// TIA Portal project "Projekt_magazyn" (V13)
// Vorlageprojekt für das Buch mit Zielsystem S7-1200

(* hardware
DEVICE "S7-1200-Station_1"  S7-1200 Station
   slot 0: "Baugruppenträger_0"  Rack  V1.0
   slot 1: "PLC_1"  CPU 1211C DC/DC/DC  6ES7 211-1AE40-0XB0  V4.1
*)

// ===== PLC "PLC_1"  CPU 1211C DC/DC/DC =====

VAR_GLOBAL   // PLC tag table "Wejścia"
   "Start" AT %I10.0 : Bool;
   "Reset" AT %I10.1 : Bool;
   "Stop" AT %I10.2 : Bool;
   "Manual" AT %I10.3 : Bool;
   "Auto" AT %I10.4 : Bool;
   "Emergency stop" AT %I10.5 : Bool;
   "Stop Baza 1" AT %I10.6 : Bool;
   "Czujnik KUKA Baza" AT %I10.7 : Bool;
   "Czujnik Baza 1" AT %I11.0 : Bool;
   "Czujnik Stop Baza" AT %I11.1 : Bool;
   "Baza gotowa" AT %I11.2 : Bool;
   "Czujnik Zacisk Baza" AT %I11.3 : Bool;
   "Stop Pokrywa 1" AT %I11.4 : Bool;
   "Czujnik KUKA Pokrywa" AT %I11.5 : Bool;
   "Czujnik Pokrywa 1" AT %I11.6 : Bool;
   "Czujnik Stop POKRYWA" AT %I11.7 : Bool;
   "Pokrywa gotowa" AT %I12.0 : Bool;
   "Czujnik Zacisk POKRYWA" AT %I12.1 : Bool;
   "Pokrywa wykryta" AT %I12.2 : Bool;
   "Moving X" AT %I12.3 : Bool;
   "Moving Z" AT %I12.4 : Bool;
   "Pos. at limit (base)" AT %I12.5 : Bool;
   "Pos. at limit (lids)" AT %I12.6 : Bool;
   "FACTORY I/O (Running)" AT %I13.0 : Bool;
   "Czujnik Sortowania" AT %ID30 : DInt;
   "Czujnik Wyjscia" AT %I13.1 : Bool;
END_VAR

VAR_GLOBAL   // PLC tag table "Wyjścia"
   "Emiter BAZA" AT %Q0.0 : Bool;
   "Baza 1" AT %Q0.1 : Bool;
   "Kuka BAZA (Start)" AT %Q0.2 : Bool;
   "Kuka BAZA (Reset)" AT %Q0.3 : Bool;
   "Kuka BAZA (Produce Base)" AT %Q0.5 : Bool;
   "Kuka BAZA (Stop)" AT %Q0.4 : Bool;
   "Baza 2" AT %Q0.6 : Bool;
   "Stop BAZA" AT %Q0.7 : Bool;
   "Baza 3" AT %Q1.0 : Bool;
   "Baza 4" AT %Q1.1 : Bool;
   "Baza 5" AT %Q1.2 : Bool;
   "Emiter POKRYWA" AT %Q1.3 : Bool;
   "Pokrywa 1" AT %Q1.4 : Bool;
   "Kuka POKRYWA (Start)" AT %Q1.5 : Bool;
   "Kuka POKRYWA (Reset)" AT %Q1.6 : Bool;
   "Kuka POKRYWA (Stop)" AT %Q1.7 : Bool;
   "Kuka POKRYWA (Produce Lids)" AT %Q2.0 : Bool;
   "Pokrywa 2" AT %Q2.1 : Bool;
   "Stop POKRYWA" AT %Q2.2 : Bool;
   "Pokrywa 3" AT %Q2.3 : Bool;
   "Pokrywa 4" AT %Q2.4 : Bool;
   "Pokrywa 5" AT %Q2.5 : Bool;
   "Baza Assembler" AT %Q2.6 : Bool;
   "Pokrywa Assembler" AT %Q2.7 : Bool;
   "Zacisk POKRYWA" AT %Q3.1 : Bool;
   "Zlap" AT %Q3.2 : Bool;
   "Podnies BAZA" AT %Q3.3 : Bool;
   "Move Z" AT %Q3.5 : Bool;
   "Move X" AT %Q3.4 : Bool;
   "tasma 1" AT %Q3.6 : Bool;
   "tasma 2" AT %Q3.7 : Bool;
   "Ramie N" AT %Q4.0 : Bool;
   "Tasma Ramie N" AT %Q4.1 : Bool;
   "Ramie Z" AT %Q4.2 : Bool;
   "Tasma Ramie Z" AT %Q4.3 : Bool;
   "Ramie I" AT %Q4.4 : Bool;
   "Tasma Ramie I" AT %Q4.5 : Bool;
   "NIEBIESKIE" AT %Q4.6 : Bool;
   "ZIELONE" AT %Q4.7 : Bool;
   "INNE" AT %Q5.0 : Bool;
   "Start light" AT %Q5.1 : Bool;
   "Reset light" AT %Q5.2 : Bool;
   "Stop light" AT %Q5.3 : Bool;
   "Zacisk BAZA" AT %Q3.0 : Bool;
   "Licznik Zielone" AT %QD34 : DInt;
   "Licznik Niebieskie" AT %QD30 : DInt;
   "Licznik Inne" AT %QD38 : DInt;
END_VAR

VAR_GLOBAL   // PLC tag table "Markery"
   "M0" AT %M0.0 : Bool;
   "M1" AT %M0.1 : Bool;
   "M2" AT %M0.2 : Bool;
   "M3" AT %M0.3 : Bool;
   "M4" AT %M0.4 : Bool;
   "M5" AT %M0.5 : Bool;
   "M6" AT %M0.6 : Bool;
   "Czujnik Sortowania w zakresie" AT %M1.4 : Bool;
   "Always False" AT %M2.0 : Bool;
END_VAR

// folder: System blocks/Program resources

DATA_BLOCK "IEC_Counter_0_DB"   // DB2
{ S7_Optimized_Access := 'FALSE' }
AUTHOR : Simatic
FAMILY : IEC
NAME : CNTR
VERSION : 1.0
// stored: InstanceOfName ?
"?"
BEGIN
END_DATA_BLOCK

DATA_BLOCK "IEC_Counter_0_DB_1"   // DB3
{ S7_Optimized_Access := 'FALSE' }
AUTHOR : Simatic
FAMILY : IEC
NAME : CNTR
VERSION : 1.0
// stored: InstanceOfName ?
"?"
BEGIN
END_DATA_BLOCK

DATA_BLOCK "IEC_Counter_0_DB_2"   // DB4
{ S7_Optimized_Access := 'FALSE' }
AUTHOR : Simatic
FAMILY : IEC
NAME : CNTR
VERSION : 1.0
// stored: InstanceOfName ?
"?"
BEGIN
END_DATA_BLOCK

// folder: (top level)

FUNCTION "MHJ-PLC-Lab-Function-S71200" : Void   // FC9000, SCL
{ S7_Optimized_Access := 'FALSE' }
VERSION : 0.1
BEGIN

   #Value:=PEEK(area := 16#82,
        dbNumber := 0,
        byteOffset := 511);
   #Value := #Value + 1;

   POKE(area := 16#82,
        dbNumber := 0,
        byteOffset := 511,
        value := #Value);

   POKE(area:=16#81,
        dbNumber:=0,
        byteOffset:=1016,
        value:=#Value_01_DW);
   POKE(area := 16#81,
        dbNumber := 0,
        byteOffset := 1020,
        value := #Value_02_DW);

   POKE(area := 16#81,
        dbNumber := 0,
        byteOffset := 511,
        value := B#16#00);

   FOR #forVal := 0 TO 120 DO
       FOR #forVal_2:=0 TO 10 DO
           #rdTimeReturn:=RD_SYS_T(#outputTime);
           #rdTimeReturn := WR_SYS_T(#outputTime);
           #rdTimeReturn := RD_SYS_T(#outputTime);
           #rdTimeReturn := WR_SYS_T(#outputTime);
       END_FOR;
       #SyncVal:= PEEK(area := 16#81,
                      dbNumber := 0,
                      byteOffset := 511);
       IF #SyncVal = #CompVal THEN
          GOTO M_1;
       END_IF;
   END_FOR;
   RETURN;

   M_1:
   POKE(area := 16#81,
        dbNumber := 0,
        byteOffset := 511,
        value := B#16#0);
END_FUNCTION

ORGANIZATION_BLOCK "Sortownia"   // OB1, LAD, ProgramCycle
TITLE = "Main Program Sweep (Cycle)"
{ S7_Optimized_Access := 'FALSE' }
VERSION : 0.1
   VAR_TEMP   // added for the SCL form of the ladder/FBD networks
      _w1 : Bool;
   END_VAR
BEGIN

REGION Network 1
   // Czujnik Sortowania (zakres wykrywania pokrywek według dokumentacji Factory IO)
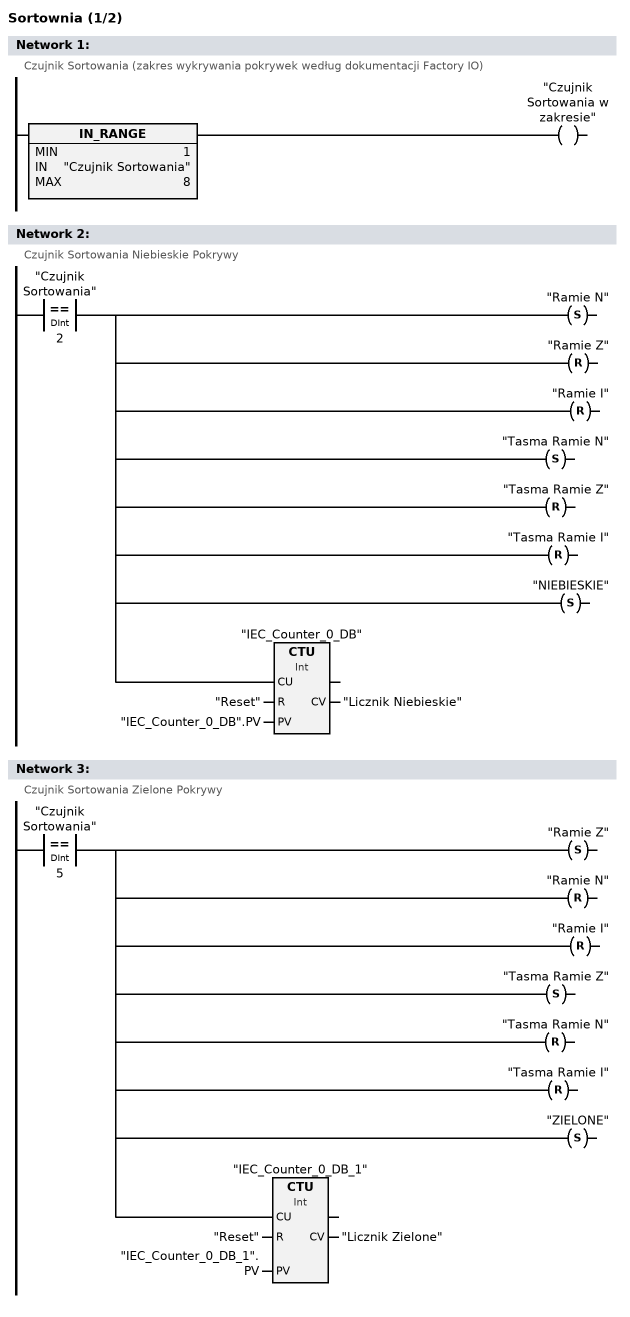
   RUNG wire#powerrail
      { S7_Templates := "SrcType := DInt" } InRange(min := 1, in := "Czujnik Sortowania", max := 8)
      Coil( "Czujnik Sortowania w zakresie" )
   END_RUNG
   // the same network as SCL:
   "Czujnik Sortowania w zakresie" := (1 <= "Czujnik Sortowania") AND ("Czujnik Sortowania" <= 8);
END_REGION

REGION Network 2
   // Czujnik Sortowania Niebieskie Pokrywy
   #_w1 := "Czujnik Sortowania" = 2;
   IF #_w1 THEN
       "Ramie N" := TRUE;
       "Ramie Z" := FALSE;
       "Ramie I" := FALSE;
       "Tasma Ramie N" := TRUE;
       "Tasma Ramie Z" := FALSE;
       "Tasma Ramie I" := FALSE;
       "NIEBIESKIE" := TRUE;
   END_IF;
   "IEC_Counter_0_DB".CTU(CU := #_w1, R := "Reset", PV := "IEC_Counter_0_DB".PV, CV => "Licznik Niebieskie");
END_REGION

REGION Network 3
   // Czujnik Sortowania Zielone Pokrywy
   #_w1 := "Czujnik Sortowania" = 5;
   IF #_w1 THEN
       "Ramie Z" := TRUE;
       "Ramie N" := FALSE;
       "Ramie I" := FALSE;
       "Tasma Ramie Z" := TRUE;
       "Tasma Ramie N" := FALSE;
       "Tasma Ramie I" := FALSE;
       "ZIELONE" := TRUE;
   END_IF;
   "IEC_Counter_0_DB_1".CTU(CU := #_w1, R := "Reset", PV := "IEC_Counter_0_DB_1".PV, CV => "Licznik Zielone");
END_REGION

REGION Network 4
   // Czujnik Sortowania Metalowe Pokrywy
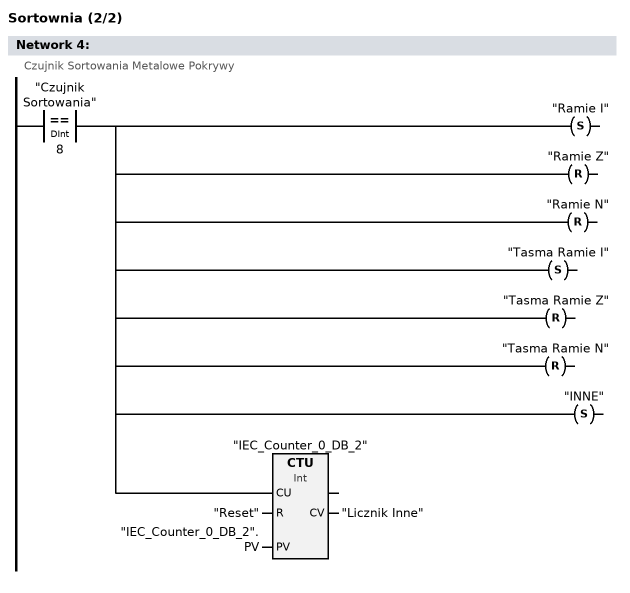
   #_w1 := "Czujnik Sortowania" = 8;
   IF #_w1 THEN
       "Ramie I" := TRUE;
       "Ramie Z" := FALSE;
       "Ramie N" := FALSE;
       "Tasma Ramie I" := TRUE;
       "Tasma Ramie Z" := FALSE;
       "Tasma Ramie N" := FALSE;
       "INNE" := TRUE;
   END_IF;
   "IEC_Counter_0_DB_2".CTU(CU := #_w1, R := "Reset", PV := "IEC_Counter_0_DB_2".PV, CV => "Licznik Inne");
END_REGION
END_ORGANIZATION_BLOCK

ORGANIZATION_BLOCK "Main 1"   // OB123, LAD, ProgramCycle
TITLE = "Main Program Sweep (Cycle)"
{ S7_Optimized_Access := 'FALSE' }
VERSION : 0.1
BEGIN

REGION Network 1
   // konfiguracja z Factory IO
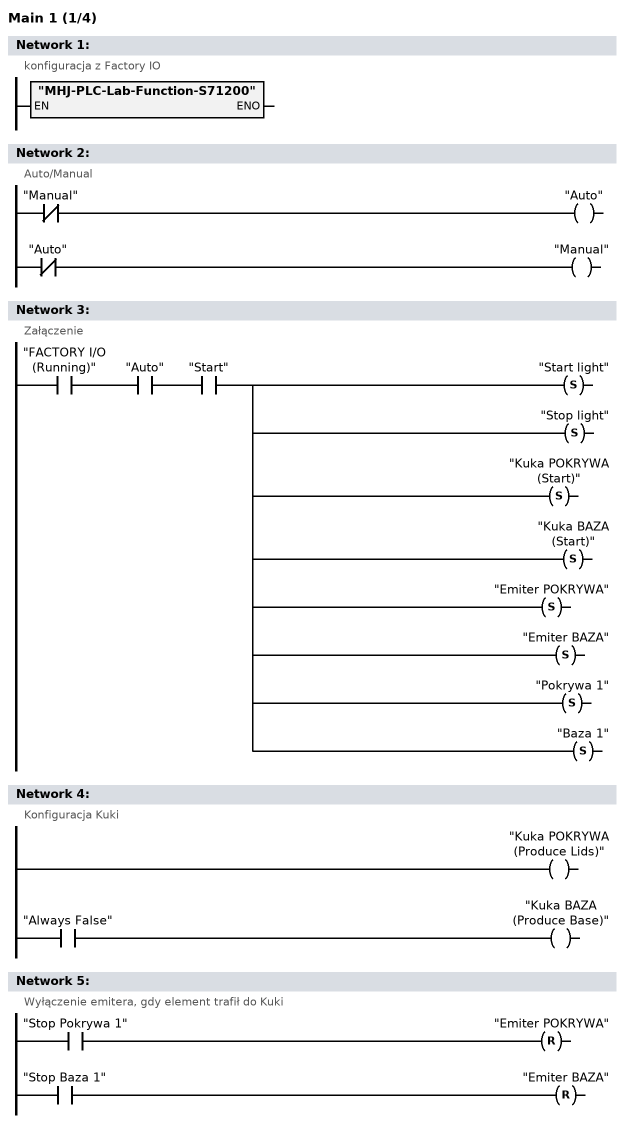
   RUNG wire#powerrail
      "MHJ-PLC-Lab-Function-S71200"()
   END_RUNG
   // the same network as SCL:
   "MHJ-PLC-Lab-Function-S71200"();
END_REGION

REGION Network 2
   // Auto/Manual
   RUNG wire#powerrail
      I_Contact( "Manual" )
      Coil( "Auto" )
   END_RUNG
   RUNG wire#powerrail
      I_Contact( "Auto" )
      Coil( "Manual" )
   END_RUNG
   // the same network as SCL:
   "Auto" := NOT "Manual";
   "Manual" := NOT "Auto";
END_REGION

REGION Network 3
   // Załączenie
   RUNG wire#powerrail
      Contact( "FACTORY I/O (Running)" )
      Contact( "Auto" )
      Contact( "Start" )
      wire#w1
      S_Coil( "Start light" )
   END_RUNG
   RUNG wire#w1
      S_Coil( "Stop light" )
   END_RUNG
   RUNG wire#w1
      S_Coil( "Kuka POKRYWA (Start)" )
   END_RUNG
   RUNG wire#w1
      S_Coil( "Kuka BAZA (Start)" )
   END_RUNG
   RUNG wire#w1
      S_Coil( "Emiter POKRYWA" )
   END_RUNG
   RUNG wire#w1
      S_Coil( "Emiter BAZA" )
   END_RUNG
   RUNG wire#w1
      S_Coil( "Pokrywa 1" )
   END_RUNG
   RUNG wire#w1
      S_Coil( "Baza 1" )
   END_RUNG
   // the same network as SCL:
   IF "FACTORY I/O (Running)" AND "Auto" AND "Start" THEN
       "Start light" := TRUE;
       "Stop light" := TRUE;
       "Kuka POKRYWA (Start)" := TRUE;
       "Kuka BAZA (Start)" := TRUE;
       "Emiter POKRYWA" := TRUE;
       "Emiter BAZA" := TRUE;
       "Pokrywa 1" := TRUE;
       "Baza 1" := TRUE;
   END_IF;
END_REGION

REGION Network 4
   // Konfiguracja Kuki
   RUNG wire#powerrail
      Coil( "Kuka POKRYWA (Produce Lids)" )
   END_RUNG
   RUNG wire#powerrail
      Contact( "Always False" )
      Coil( "Kuka BAZA (Produce Base)" )
   END_RUNG
   // the same network as SCL:
   "Kuka POKRYWA (Produce Lids)" := TRUE;
   "Kuka BAZA (Produce Base)" := "Always False";
END_REGION

REGION Network 5
   // Wyłączenie emitera, gdy element trafił do Kuki
   RUNG wire#powerrail
      Contact( "Stop Pokrywa 1" )
      R_Coil( "Emiter POKRYWA" )
   END_RUNG
   RUNG wire#powerrail
      Contact( "Stop Baza 1" )
      R_Coil( "Emiter BAZA" )
   END_RUNG
   // the same network as SCL:
   IF "Stop Pokrywa 1" THEN "Emiter POKRYWA" := FALSE; END_IF;
   IF "Stop Baza 1" THEN "Emiter BAZA" := FALSE; END_IF;
END_REGION

REGION Network 6
   // Sterowanie taśmą i Stop Blade po wykryciu elementu
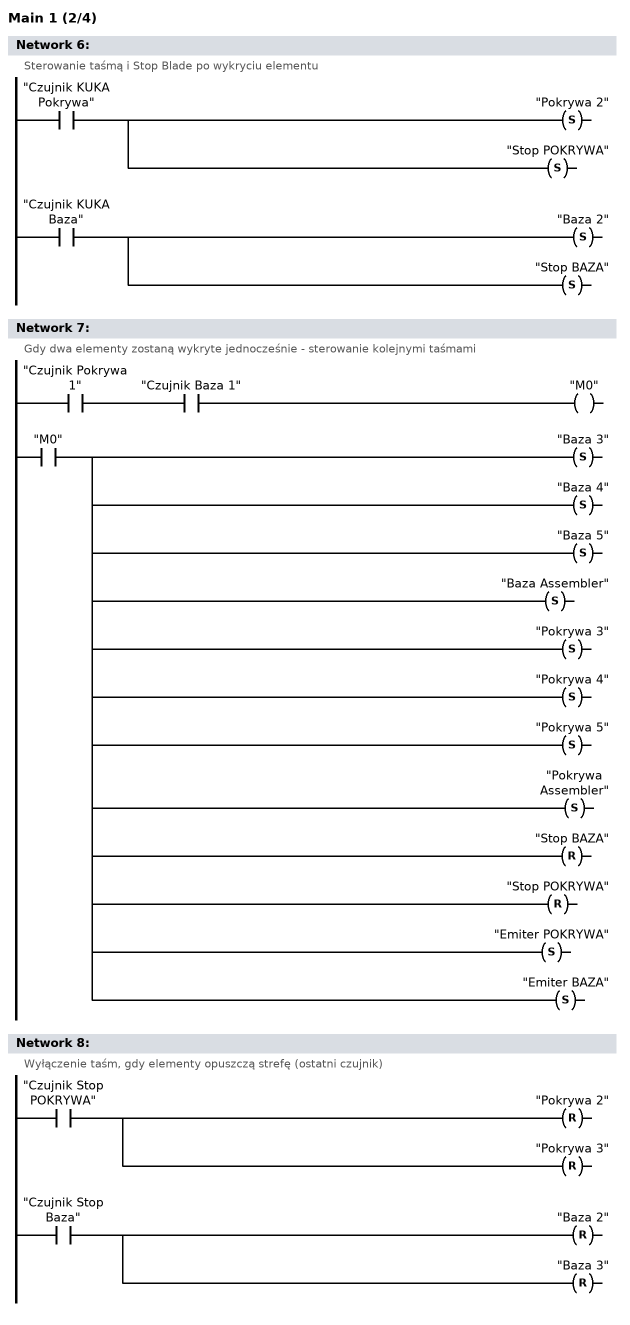
   RUNG wire#powerrail
      Contact( "Czujnik KUKA Pokrywa" )
      wire#w1
      S_Coil( "Pokrywa 2" )
   END_RUNG
   RUNG wire#w1
      S_Coil( "Stop POKRYWA" )
   END_RUNG
   RUNG wire#powerrail
      Contact( "Czujnik KUKA Baza" )
      wire#w2
      S_Coil( "Baza 2" )
   END_RUNG
   RUNG wire#w2
      S_Coil( "Stop BAZA" )
   END_RUNG
   // the same network as SCL:
   IF "Czujnik KUKA Pokrywa" THEN
       "Pokrywa 2" := TRUE;
       "Stop POKRYWA" := TRUE;
   END_IF;
   IF "Czujnik KUKA Baza" THEN
       "Baza 2" := TRUE;
       "Stop BAZA" := TRUE;
   END_IF;
END_REGION

REGION Network 7
   // Gdy dwa elementy zostaną wykryte jednocześnie - sterowanie kolejnymi taśmami
   RUNG wire#powerrail
      Contact( "Czujnik Pokrywa 1" )
      Contact( "Czujnik Baza 1" )
      Coil( "M0" )
   END_RUNG
   RUNG wire#powerrail
      Contact( "M0" )
      wire#w1
      S_Coil( "Baza 3" )
   END_RUNG
   RUNG wire#w1
      S_Coil( "Baza 4" )
   END_RUNG
   RUNG wire#w1
      S_Coil( "Baza 5" )
   END_RUNG
   RUNG wire#w1
      S_Coil( "Baza Assembler" )
   END_RUNG
   RUNG wire#w1
      S_Coil( "Pokrywa 3" )
   END_RUNG
   RUNG wire#w1
      S_Coil( "Pokrywa 4" )
   END_RUNG
   RUNG wire#w1
      S_Coil( "Pokrywa 5" )
   END_RUNG
   RUNG wire#w1
      S_Coil( "Pokrywa Assembler" )
   END_RUNG
   RUNG wire#w1
      R_Coil( "Stop BAZA" )
   END_RUNG
   RUNG wire#w1
      R_Coil( "Stop POKRYWA" )
   END_RUNG
   RUNG wire#w1
      S_Coil( "Emiter POKRYWA" )
   END_RUNG
   RUNG wire#w1
      S_Coil( "Emiter BAZA" )
   END_RUNG
   // the same network as SCL:
   "M0" := "Czujnik Pokrywa 1" AND "Czujnik Baza 1";
   IF "M0" THEN
       "Baza 3" := TRUE;
       "Baza 4" := TRUE;
       "Baza 5" := TRUE;
       "Baza Assembler" := TRUE;
       "Pokrywa 3" := TRUE;
       "Pokrywa 4" := TRUE;
       "Pokrywa 5" := TRUE;
       "Pokrywa Assembler" := TRUE;
       "Stop BAZA" := FALSE;
       "Stop POKRYWA" := FALSE;
       "Emiter POKRYWA" := TRUE;
       "Emiter BAZA" := TRUE;
   END_IF;
END_REGION

REGION Network 8
   // Wyłączenie taśm, gdy elementy opuszczą strefę (ostatni czujnik)
   RUNG wire#powerrail
      Contact( "Czujnik Stop POKRYWA" )
      wire#w1
      R_Coil( "Pokrywa 2" )
   END_RUNG
   RUNG wire#w1
      R_Coil( "Pokrywa 3" )
   END_RUNG
   RUNG wire#powerrail
      Contact( "Czujnik Stop Baza" )
      wire#w2
      R_Coil( "Baza 2" )
   END_RUNG
   RUNG wire#w2
      R_Coil( "Baza 3" )
   END_RUNG
   // the same network as SCL:
   IF "Czujnik Stop POKRYWA" THEN
       "Pokrywa 2" := FALSE;
       "Pokrywa 3" := FALSE;
   END_IF;
   IF "Czujnik Stop Baza" THEN
       "Baza 2" := FALSE;
       "Baza 3" := FALSE;
   END_IF;
END_REGION

REGION Network 9
   // STOP
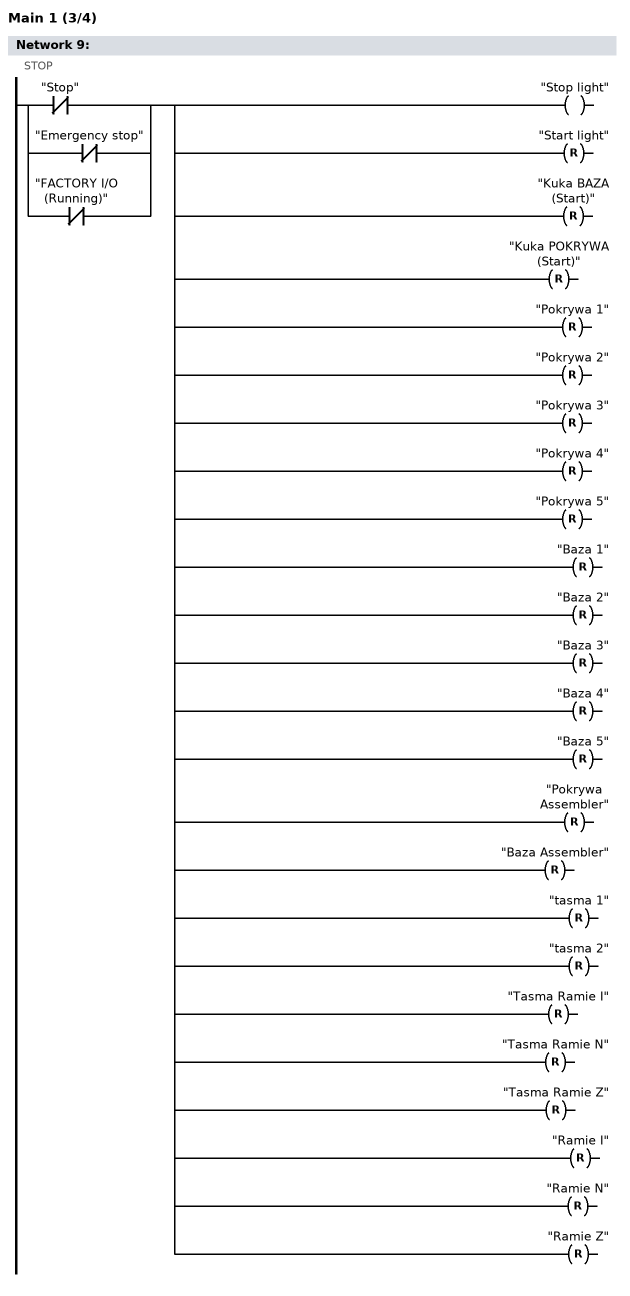
   RUNG wire#powerrail
      I_Contact( "Stop" )
      wire#w1
      Coil( "Stop light" )
   END_RUNG
   RUNG wire#powerrail
      I_Contact( "Emergency stop" )
   END_RUNG wire#w1
   RUNG wire#powerrail
      I_Contact( "FACTORY I/O (Running)" )
   END_RUNG wire#w1
   RUNG wire#w1
      R_Coil( "Start light" )
   END_RUNG
   RUNG wire#w1
      R_Coil( "Kuka BAZA (Start)" )
   END_RUNG
   RUNG wire#w1
      R_Coil( "Kuka POKRYWA (Start)" )
   END_RUNG
   RUNG wire#w1
      R_Coil( "Pokrywa 1" )
   END_RUNG
   RUNG wire#w1
      R_Coil( "Pokrywa 2" )
   END_RUNG
   RUNG wire#w1
      R_Coil( "Pokrywa 3" )
   END_RUNG
   RUNG wire#w1
      R_Coil( "Pokrywa 4" )
   END_RUNG
   RUNG wire#w1
      R_Coil( "Pokrywa 5" )
   END_RUNG
   RUNG wire#w1
      R_Coil( "Baza 1" )
   END_RUNG
   RUNG wire#w1
      R_Coil( "Baza 2" )
   END_RUNG
   RUNG wire#w1
      R_Coil( "Baza 3" )
   END_RUNG
   RUNG wire#w1
      R_Coil( "Baza 4" )
   END_RUNG
   RUNG wire#w1
      R_Coil( "Baza 5" )
   END_RUNG
   RUNG wire#w1
      R_Coil( "Pokrywa Assembler" )
   END_RUNG
   RUNG wire#w1
      R_Coil( "Baza Assembler" )
   END_RUNG
   RUNG wire#w1
      R_Coil( "tasma 1" )
   END_RUNG
   RUNG wire#w1
      R_Coil( "tasma 2" )
   END_RUNG
   RUNG wire#w1
      R_Coil( "Tasma Ramie I" )
   END_RUNG
   RUNG wire#w1
      R_Coil( "Tasma Ramie N" )
   END_RUNG
   RUNG wire#w1
      R_Coil( "Tasma Ramie Z" )
   END_RUNG
   RUNG wire#w1
      R_Coil( "Ramie I" )
   END_RUNG
   RUNG wire#w1
      R_Coil( "Ramie N" )
   END_RUNG
   RUNG wire#w1
      R_Coil( "Ramie Z" )
   END_RUNG
   // the same network as SCL:
   "Stop light" := NOT "Stop" OR NOT "Emergency stop" OR NOT "FACTORY I/O (Running)";
   IF "Stop light" THEN
       "Start light" := FALSE;
       "Kuka BAZA (Start)" := FALSE;
       "Kuka POKRYWA (Start)" := FALSE;
       "Pokrywa 1" := FALSE;
       "Pokrywa 2" := FALSE;
       "Pokrywa 3" := FALSE;
       "Pokrywa 4" := FALSE;
       "Pokrywa 5" := FALSE;
       "Baza 1" := FALSE;
       "Baza 2" := FALSE;
       "Baza 3" := FALSE;
       "Baza 4" := FALSE;
       "Baza 5" := FALSE;
       "Pokrywa Assembler" := FALSE;
       "Baza Assembler" := FALSE;
       "tasma 1" := FALSE;
       "tasma 2" := FALSE;
       "Tasma Ramie I" := FALSE;
       "Tasma Ramie N" := FALSE;
       "Tasma Ramie Z" := FALSE;
       "Ramie I" := FALSE;
       "Ramie N" := FALSE;
       "Ramie Z" := FALSE;
   END_IF;
END_REGION

REGION Network 10
   // Reset
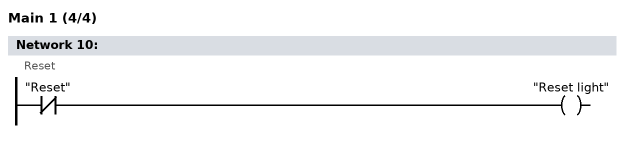
   RUNG wire#powerrail
      I_Contact( "Reset" )
      Coil( "Reset light" )
   END_RUNG
   // the same network as SCL:
   "Reset light" := NOT "Reset";
END_REGION
END_ORGANIZATION_BLOCK

ORGANIZATION_BLOCK "AssemblerKroki"   // OB125, LAD, ProgramCycle
TITLE = "Main Program Sweep (Cycle)"
{ S7_Optimized_Access := 'FALSE' }
VERSION : 0.1
   VAR_TEMP   // added for the SCL form of the ladder/FBD networks
      _w1 : Bool;
      _w2 : Bool;
      _w3 : Bool;
      _w4 : Bool;
      _w5 : Bool;
   END_VAR
BEGIN

REGION Network 1
   // Zaciskanie Pokrywy
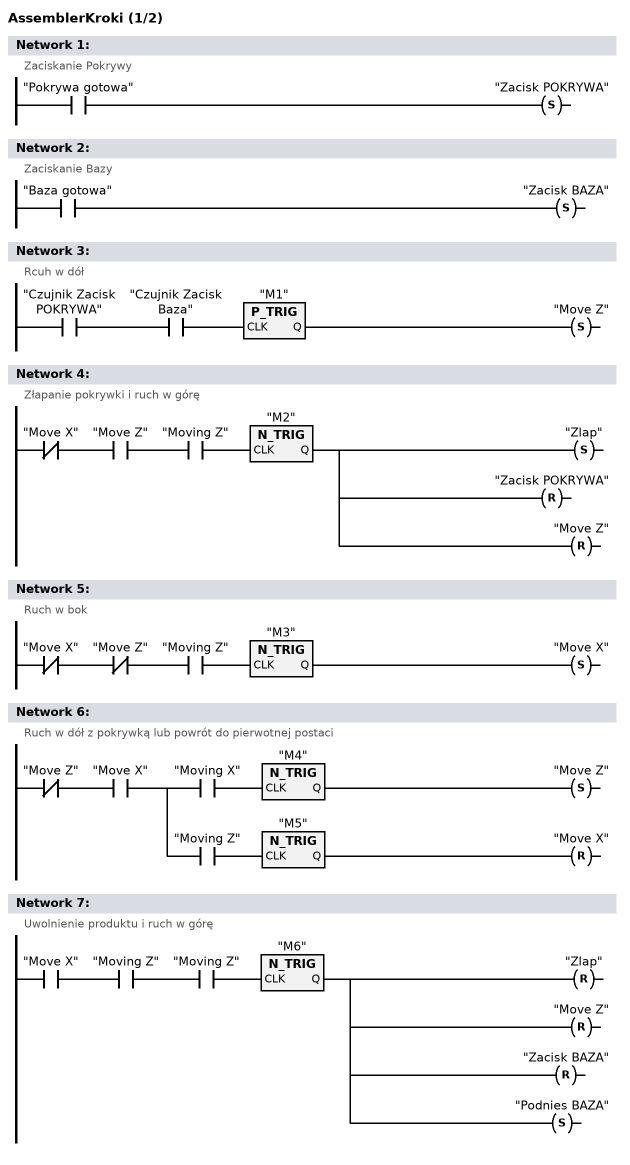
   RUNG wire#powerrail
      Contact( "Pokrywa gotowa" )
      S_Coil( "Zacisk POKRYWA" )
   END_RUNG
   // the same network as SCL:
   IF "Pokrywa gotowa" THEN "Zacisk POKRYWA" := TRUE; END_IF;
END_REGION

REGION Network 2
   // Zaciskanie Bazy
   RUNG wire#powerrail
      Contact( "Baza gotowa" )
      S_Coil( "Zacisk BAZA" )
   END_RUNG
   // the same network as SCL:
   IF "Baza gotowa" THEN "Zacisk BAZA" := TRUE; END_IF;
END_REGION

REGION Network 3
   // Rcuh w dół
   RUNG wire#powerrail
      Contact( "Czujnik Zacisk POKRYWA" )
      Contact( "Czujnik Zacisk Baza" )
      P_Trig( "M1" )
      S_Coil( "Move Z" )
   END_RUNG
   // the same network as SCL:
   #_w1 := "Czujnik Zacisk POKRYWA" AND "Czujnik Zacisk Baza";
   #_w2 := #_w1 AND NOT "M1";   // rising edge
   "M1" := #_w1;
   IF #_w2 THEN "Move Z" := TRUE; END_IF;
END_REGION

REGION Network 4
   // Złapanie pokrywki i ruch w górę
   RUNG wire#powerrail
      I_Contact( "Move X" )
      Contact( "Move Z" )
      Contact( "Moving Z" )
      N_Trig( "M2" )
      wire#w1
      S_Coil( "Zlap" )
   END_RUNG
   RUNG wire#w1
      R_Coil( "Zacisk POKRYWA" )
   END_RUNG
   RUNG wire#w1
      R_Coil( "Move Z" )
   END_RUNG
   // the same network as SCL:
   #_w1 := NOT "Move X" AND "Move Z" AND "Moving Z";
   #_w2 := NOT #_w1 AND "M2";   // falling edge
   "M2" := #_w1;
   IF #_w2 THEN
       "Zlap" := TRUE;
       "Zacisk POKRYWA" := FALSE;
       "Move Z" := FALSE;
   END_IF;
END_REGION

REGION Network 5
   // Ruch w bok
   RUNG wire#powerrail
      I_Contact( "Move X" )
      I_Contact( "Move Z" )
      Contact( "Moving Z" )
      N_Trig( "M3" )
      S_Coil( "Move X" )
   END_RUNG
   // the same network as SCL:
   #_w1 := NOT "Move X" AND NOT "Move Z" AND "Moving Z";
   #_w2 := NOT #_w1 AND "M3";   // falling edge
   "M3" := #_w1;
   IF #_w2 THEN "Move X" := TRUE; END_IF;
END_REGION

REGION Network 6
   // Ruch w dół z pokrywką lub powrót do pierwotnej postaci
   RUNG wire#powerrail
      I_Contact( "Move Z" )
      Contact( "Move X" )
      wire#w1
      Contact( "Moving X" )
      N_Trig( "M4" )
      S_Coil( "Move Z" )
   END_RUNG
   RUNG wire#w1
      Contact( "Moving Z" )
      N_Trig( "M5" )
      R_Coil( "Move X" )
   END_RUNG
   // the same network as SCL:
   #_w1 := NOT "Move Z" AND "Move X";
   #_w2 := #_w1 AND "Moving X";
   #_w3 := NOT #_w2 AND "M4";   // falling edge
   "M4" := #_w2;
   IF #_w3 THEN "Move Z" := TRUE; END_IF;
   #_w4 := #_w1 AND "Moving Z";
   #_w5 := NOT #_w4 AND "M5";   // falling edge
   "M5" := #_w4;
   IF #_w5 THEN "Move X" := FALSE; END_IF;
END_REGION

REGION Network 7
   // Uwolnienie produktu i ruch w górę
   RUNG wire#powerrail
      Contact( "Move X" )
      Contact( "Moving Z" )
      Contact( "Moving Z" )
      N_Trig( "M6" )
      wire#w1
      R_Coil( "Zlap" )
   END_RUNG
   RUNG wire#w1
      R_Coil( "Move Z" )
   END_RUNG
   RUNG wire#w1
      R_Coil( "Zacisk BAZA" )
   END_RUNG
   RUNG wire#w1
      S_Coil( "Podnies BAZA" )
   END_RUNG
   // the same network as SCL:
   #_w1 := "Move X" AND "Moving Z" AND "Moving Z";
   #_w2 := NOT #_w1 AND "M6";   // falling edge
   "M6" := #_w1;
   IF #_w2 THEN
       "Zlap" := FALSE;
       "Move Z" := FALSE;
       "Zacisk BAZA" := FALSE;
       "Podnies BAZA" := TRUE;
   END_IF;
END_REGION

REGION Network 8
   // Uruchomienie taśm i ustawienie blokady
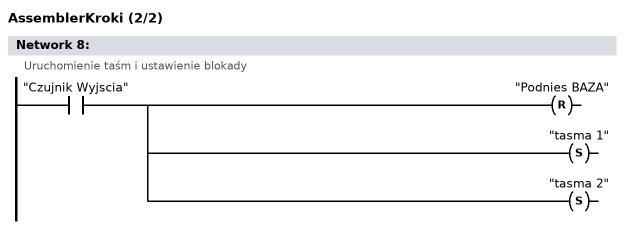
   RUNG wire#powerrail
      Contact( "Czujnik Wyjscia" )
      wire#w1
      R_Coil( "Podnies BAZA" )
   END_RUNG
   RUNG wire#w1
      S_Coil( "tasma 1" )
   END_RUNG
   RUNG wire#w1
      S_Coil( "tasma 2" )
   END_RUNG
   // the same network as SCL:
   IF "Czujnik Wyjscia" THEN
       "Podnies BAZA" := FALSE;
       "tasma 1" := TRUE;
       "tasma 2" := TRUE;
   END_IF;
END_REGION
END_ORGANIZATION_BLOCK